PROGRAM MAP_IN
VAR
  byPassMapping     : BOOL;

  uTransportCtrl    : U_XTS_TRANSPORT_CTRL;
  uStationCtrl      : U_STATION_CTRL;
END_VAR


IF NOT (byPassMapping)
THEN
  memcpy(ADR(GVL_XTS.XtsTransportCtrl),   ADR(uTransportCtrl),  SIZEOF(ST_XTS_TRANSPORT_CTRL));
  memcpy(ADR(GVL_XTS.StationCtrl),        ADR(uStationCtrl),    SIZEOF(uStationCtrl));
END_IF

END_PROGRAM

(* stored: Version 1.1.0.1, ProductVersion 3.1.4024.12
   POU MAP_IN: Id {2f0d255c-74ed-4d54-a393-b49ffab3376d}, SpecialFunc None *)
